{attribute addProperty BoxType "AX8620-0000-0026"}
{attribute addProperty Id "PSM_StatuswordAT %I*PSM_Statusword_32E7AA9A1620WcStateAT %I*WcState_F855686C1620InfoDataAT %I*InfoData_0BDED7BF144180"}
{attribute addProperty CRC "914595954"}
{attribute addProperty SizeInBites "176"}
{attribute addProperty SizeInBytes "22"}
TYPE AX8620_86637E7C :
STRUCT
	{attribute addProperty Name "PSM_Statusword"}
	PSM_Statusword : PSM_Statusword_32E7AA9A;
	{attribute addProperty Name "WcState"}
	WcState : WcState_F855686C;
	{attribute addProperty Name "InfoData"}
	InfoData : InfoData_0BDED7BF;
END_STRUCT
END_TYPE

(* stored: Version 1.2.0.0, ProductVersion 3.1.4024.9
   DUT AX8620_86637E7C: Id {679a1be3-0241-49ce-823c-7db09aedce4a} *)
